FUNCTION_BLOCK L2_PlatoDivisor_SFC EXTENDS L1_ControllerBase_SFC

VAR_INPUT 					// Sensores y comandos
	d0  		: BOOL; 
END_VAR

VAR_OUTPUT					// Actuadores
	D_1 		: BOOL; 
    E_1 		: BOOL; 
END_VAR

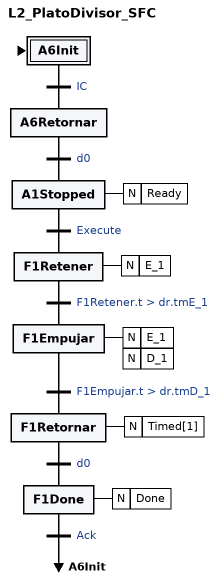
INITIAL_STEP A6Init:
END_STEP
TRANSITION FROM A6Init TO A6Retornar
    := IC;
END_TRANSITION
STEP A6Retornar:
END_STEP
TRANSITION FROM A6Retornar TO A1Stopped
    := d0;
END_TRANSITION
STEP A1Stopped:
    Ready(N);
END_STEP
TRANSITION FROM A1Stopped TO F1Retener
    := Execute;
END_TRANSITION
STEP F1Retener:
    E_1(N);
END_STEP
TRANSITION FROM F1Retener TO F1Empujar
    := F1Retener.t > dr.tmE_1;
END_TRANSITION
STEP F1Empujar:
    E_1(N);
    D_1(N);
END_STEP
TRANSITION FROM F1Empujar TO F1Retornar
    := F1Empujar.t > dr.tmD_1;
END_TRANSITION
STEP F1Retornar:
    Timed[1](N);
END_STEP
TRANSITION FROM F1Retornar TO F1Done
    := d0;
END_TRANSITION
STEP F1Done:
    Done(N);
END_STEP
TRANSITION FROM F1Done TO A6Init
    := Ack;
END_TRANSITION

END_FUNCTION_BLOCK

(* stored: Version 1.1.0.1, ProductVersion 3.1.4024.11
   POU L2_PlatoDivisor_SFC: Id {780d8d1f-d39e-46b4-929b-6b9a28c712e1}, SpecialFunc None *)
